(* PLC project Unnamed, Unknown Unnamed 1 *)
(* stored: creationDateTime 2025-02-17T01:13:19, modificationDateTime 2025-04-06T13:02:39 *)

PROGRAM ex03
  VAR
    NS_red AT %QX100.0 : BOOL;
    NS_yellow AT %QX100.1 : BOOL;
    NS_green AT %QX100.2 : BOOL;
    EW_red AT %QX0.0 : BOOL := true;
    EW_yellow AT %QX0.1 : BOOL;
    EW_green AT %QX0.2 : BOOL;
    Time_NS_green AT %MW0 : INT;
    Time_NS_yellow AT %MW1 : INT;
    Time_NS_red AT %MW2 : INT;
    Time_EW_green AT %MW3 : INT;
    Time_EW_yellow AT %MW4 : INT;
    Time_EW_red AT %MW5 : INT;
  END_VAR
  VAR
    TON0 : TON;
    TON1 : TON;
    TON2 : TON;
    TON3 : TON;
  END_VAR
  VAR  (* added by the conversion: wires and edge detectors of the diagram *)
    _SUB37_OUT : INT;
    _SUB74_OUT : INT;
  END_VAR

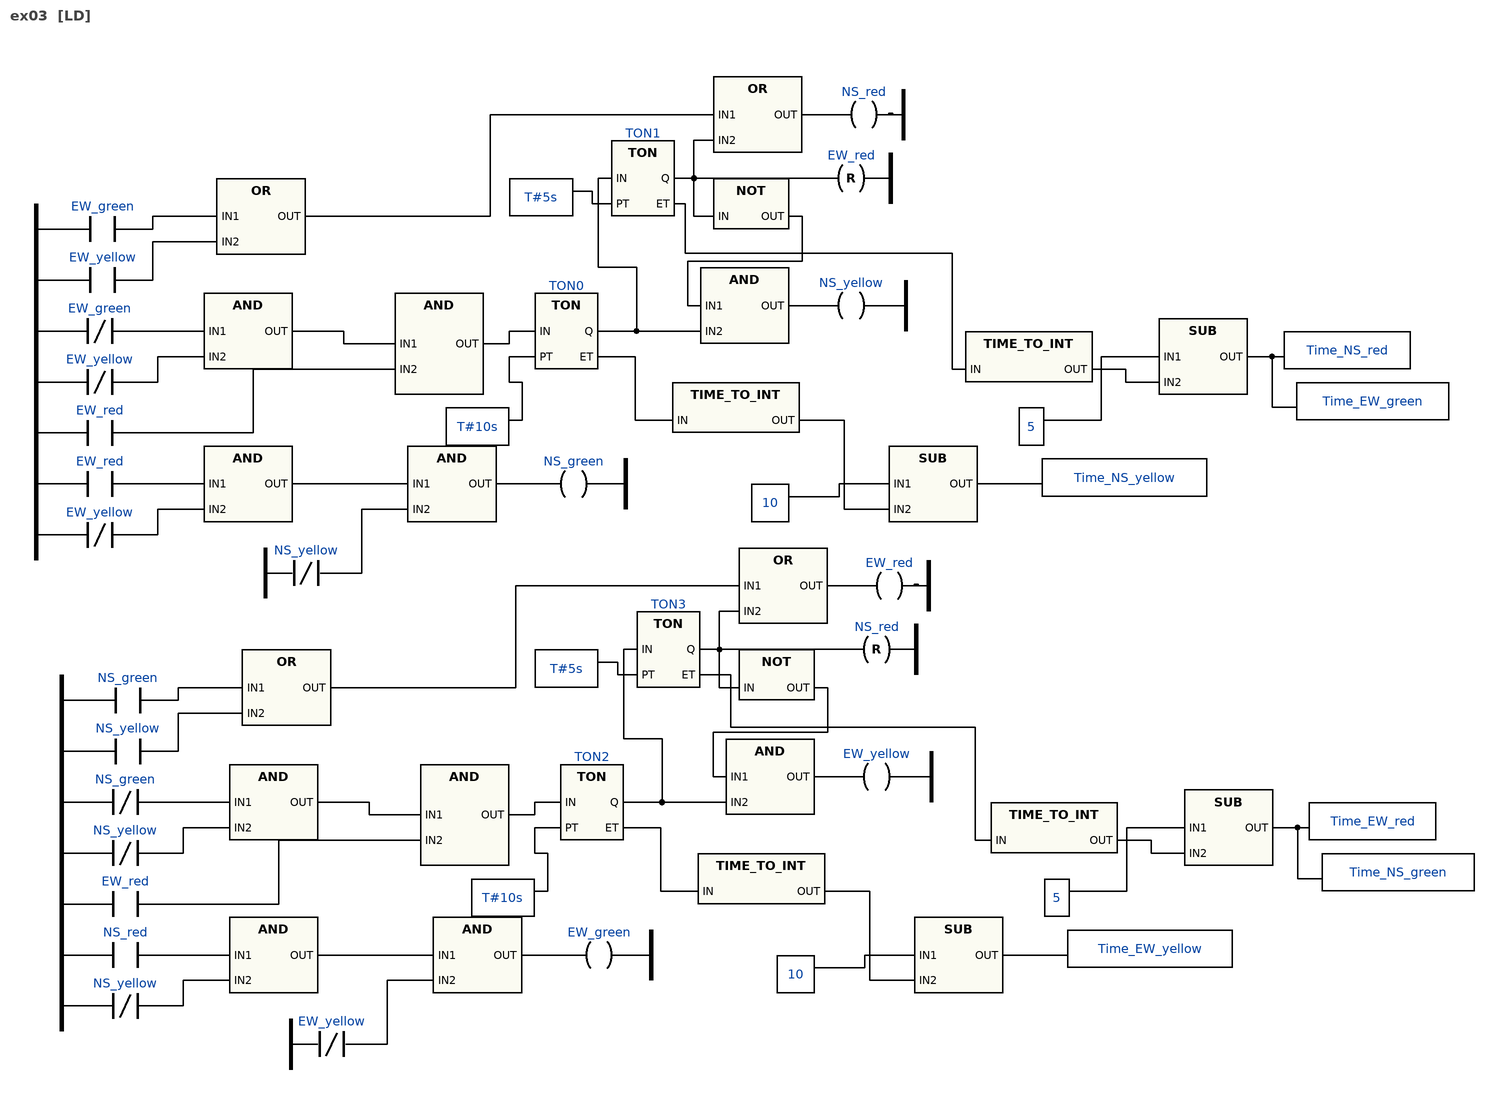
(* LD diagram, written out as Structured Text *)
NS_green := EW_red AND NOT EW_yellow AND NOT NS_yellow;
TON0(IN := NOT EW_green AND NOT EW_yellow AND EW_red, PT := T#10s);
TON1(IN := TON0.Q, PT := T#5s);
NS_yellow := NOT TON1.Q AND TON0.Q;
NS_red := EW_green OR EW_yellow OR TON1.Q;
IF TON1.Q THEN EW_red := FALSE; END_IF;
_SUB37_OUT := 5 - TIME_TO_INT(TON1.ET);
Time_NS_red := _SUB37_OUT;
Time_NS_yellow := 10 - TIME_TO_INT(TON0.ET);
Time_EW_green := _SUB37_OUT;
EW_green := NS_red AND NOT NS_yellow AND NOT EW_yellow;
TON2(IN := NOT NS_green AND NOT NS_yellow AND EW_red, PT := T#10s);
TON3(IN := TON2.Q, PT := T#5s);
EW_yellow := NOT TON3.Q AND TON2.Q;
EW_red := NS_green OR NS_yellow OR TON3.Q;
IF TON3.Q THEN NS_red := FALSE; END_IF;
_SUB74_OUT := 5 - TIME_TO_INT(TON3.ET);
Time_EW_red := _SUB74_OUT;
Time_EW_yellow := 10 - TIME_TO_INT(TON2.ET);
Time_NS_green := _SUB74_OUT;
END_PROGRAM

CONFIGURATION Config0
  RESOURCE Res0 ON PLC
    TASK task0(INTERVAL := T#20ms, PRIORITY := 0);
    PROGRAM instance0 WITH task0 : ex03;
  END_RESOURCE
END_CONFIGURATION
